Staubli VAL3: remErrBufferAdd.pgx

program remErrBufferAdd(string& sErrMessage[] (dimensions=1))
begin
  //Add an error message to the error buffer
  //Used for errors that may happen long after a command is called
  //e.g. used for end of movement errors because we can't stop the
  //  IOC to wait for them
  //
  logMsg("call remErrBufferAdd")
  sErrBuffer[nErrNext]=sErrMessage
  if nErrNext==nErrBufferSize
    nErrNext=0
  else
    nErrNext=nErrNext+1
  endIf
end
